PROGRAM MAIN
VAR
END_VAR

P_MBus();

END_PROGRAM

(* stored: Version 1.1.0.1, ProductVersion 3.1.4024.6
   POU MAIN: Id {9ddaf94b-b05e-4a9f-be69-74ff74d59ee3}, SpecialFunc None *)
